(* PLC project PLC, Beckhoff Automation GmbH TwinCAT PLC Control 3.5.13.21 *)
(* stored: creationDateTime 2024-02-17T22:42:34.5485017, modificationDateTime 2024-02-17T22:42:34.5485017 *)

TYPE LPResource :
STRUCT
	output: LPOutput;
	config: LPConfig;
	status: LPStatus;
END_STRUCT
END_TYPE
